FUNCTION_BLOCK FB_StrukturieterText
VAR_INPUT
END_VAR
VAR_OUTPUT
END_VAR
VAR
	nCounter: INT := 0;
	nCounterSav: INT := 0;
	reCount	: R_TRIG;
	ForceCheck	: BOOL;
	Ergebnis : INT ;
	Wert1	: INT;
	Wert2	: INT;
	Motor1	:BOOL;
	Motor2	:BOOL;
	Zylinder:BOOL;
	Zylinder2:BOOL;
	step:int;
	
	Bedingung: BOOL;
	Anweisungen	:BOOL;
	Anweisungen2: BOOL;
	Anweisungen3: BOOL;
END_VAR







Ergebnis := Wert1 + Wert2;


IF Bedingung THEN
	Anweisungen;
ELSIF
	Anweisungen2;
ELSE
	Anweisungen3;
END_IF





IF Bedingung THEN
	Anweisungen;
ELSIF
	Anweisungsblock2;
ELSE
	Anweisung
END_IF













CASE step OF	
	1:	Motor1:= TRUE;
		Motor2:= FALSE;
		
	2,7:	Motor1:= FALSE;
			Motor2:= TRUE;
		
	8..12:	Motor1:= TRUE;
			Motor2:= TRUE;
ELSE
		Motor1:= FALSE;
		Motor2:= FALSE;
END_CASE












nCounter := 5000;
nCounter := nCounter + 1;
nCounter := nCounter + 1;
nCounter := nCounter + 1;
nCounter := nCounter + 1;
nCounter := nCounter + 1;
nCounter := nCounter + 1;
nCounter := nCounter + 1;

//IF nCounter = 600 THEN 
//	ForceCheck := TRUE;
//ELSE
//	ForceCheck := FALSE;
//END_IF

reCount(CLK:=PRG_TaktGen.fb_Taktmerker.Takt_1s);
IF reCount.Q THEN
	nCounter := nCounter + 1;
	nCounter := nCounter + 1;
	nCounter := nCounter + 1;
	nCounter := nCounter + 1;
	nCounter := nCounter + 1;
	nCounter := nCounter + 1;
	nCounter := nCounter + 1;
	nCounterSav := nCounter;
	
END_IF

nCounter := nCounter;
IF NOT PRG_TaktGen.fb_Taktmerker.Takt_1s THEN
	nCounterSav := 0;
END_IF

END_FUNCTION_BLOCK

(* stored: Version 1.1.0.1, ProductVersion 3.1.4024.12
   POU FB_StrukturieterText: Id {b7d63741-9653-4ae0-a831-49d06c4ff234}, SpecialFunc None *)
